FUNCTION ModuloLREAL : LREAL
VAR_INPUT
	divident : LREAL;
	modulus : LREAL;
END_VAR

ModuloLREAL := divident - modulus * FLOOR(divident / modulus);

END_FUNCTION

(* stored: Version 1.1.0.1
   POU ModuloLREAL: Id {49038c5a-4f9c-05e8-19b7-02e574464d39}, SpecialFunc None *)
